LIN {X 0,Y 79.214,Z 378.176,A -85,B 0,C 180,E1 -30939.921,E2 -30939.921} C_VEL
LIN {X 0,Y 81.535,Z 365.2,A -85,B 0,C 180,E1 -30940.229,E2 -30940.229} C_VEL
LIN {X 0,Y 82.563,Z 356.649,A -85,B 0,C 180,E1 -30940.524,E2 -30940.524} C_VEL
LIN {X 0,Y 82.095,Z 354.312,A -85,B 0,C 180,E1 -30944.218,E2 -30944.218} C_VEL
LIN {X 0,Y 81.886,Z 351.905,A -85,B 0,C 180,E1 -30950.139,E2 -30950.139} C_VEL
LIN {X 0,Y 81.95,Z 352.015,A -85,B 0,C 180,E1 -30953.705,E2 -30953.705} C_VEL
LIN {X 0,Y 82.216,Z 354.524,A -85,B 0,C 180,E1 -30958.491,E2 -30958.491} C_VEL
LIN {X 0,Y 82.607,Z 356.769,A -85,B 0,C 180,E1 -30961.538,E2 -30961.538} C_VEL
LIN {X 0,Y 80.054,Z 374.634,A -85,B 0,C 180,E1 -30961.987,E2 -30961.987} C_VEL
LIN {X 0,Y 76.93,Z 387.122,A -85,B 0,C 180,E1 -30962.346,E2 -30962.346} C_VEL
LIN {X 0,Y 72.584,Z 399.313,A -85,B 0,C 180,E1 -30963.156,E2 -30963.156} C_VEL
LIN {X 0,Y 66.925,Z 411.041,A -85,B 0,C 180,E1 -30963.978,E2 -30963.978} C_VEL
LIN {X 0,Y 62.589,Z 418.476,A -85,B 0,C 180,E1 -30964.782,E2 -30964.782} C_VEL
LIN {X 0,Y 55.7,Z 428.368,A -85,B 0,C 180,E1 -30966.498,E2 -30966.498} C_VEL
LIN {X 0,Y 49.71,Z 435.606,A -85,B 0,C 180,E1 -30968.267,E2 -30968.267} C_VEL
LIN {X 0,Y 41.286,Z 444.313,A -85,B 0,C 180,E1 -30971.836,E2 -30971.836} C_VEL
LIN {X 0,Y 31.466,Z 452.724,A -85,B 0,C 180,E1 -30978.346,E2 -30978.346} C_VEL
LIN {X 0,Y 22.335,Z 459.473,A -85,B 0,C 180,E1 -30990.091,E2 -30990.091} C_VEL
LIN {X 0,Y 14.338,Z 465.618,A -85,B 0,C 180,E1 -31020.66,E2 -31020.66} C_VEL
LIN {X 0,Y 12.95,Z 468.35,A -85,B 0,C 180,E1 -31050.01,E2 -31050.01} C_VEL
LIN {X 0,Y 14.464,Z 470.587,A -85,B 0,C 180,E1 -31079.082,E2 -31079.082} C_VEL
LIN {X 0,Y 18.52,Z 472.391,A -85,B 0,C 180,E1 -31099.384,E2 -31099.384} C_VEL
LIN {X 0,Y 30.065,Z 474.714,A -85,B 0,C 180,E1 -31119.245,E2 -31119.245} C_VEL
LIN {X 0,Y 43.205,Z 475.536,A -85,B 0,C 180,E1 -31127.436,E2 -31127.436} C_VEL
LIN {X 0,Y 49.975,Z 475.374,A -85,B 0,C 180,E1 -31129.886,E2 -31129.886} C_VEL
LIN {X 0,Y 52.842,Z 475.146,A -85,B 0,C 180,E1 -31132.323,E2 -31132.323} C_VEL
LIN {X 0,Y 42.273,Z 475.423,A -85,B 0,C 180,E1 -31136.005,E2 -31136.005} C_VEL
LIN {X 0,Y 34.947,Z 475.052,A -85,B 0,C 180,E1 -31139.948,E2 -31139.948} C_VEL
LIN {X 0,Y 28.242,Z 474.29,A -85,B 0,C 180,E1 -31145.454,E2 -31145.454} C_VEL
LIN {X 0,Y 18.34,Z 472.097,A -85,B 0,C 180,E1 -31162.424,E2 -31162.424} C_VEL
LIN {X 0,Y 12.711,Z 469.162,A -85,B 0,C 180,E1 -31196.422,E2 -31196.422} C_VEL
LIN {X 0,Y 14.539,Z 464.821,A -85,B 0,C 180,E1 -31245.295,E2 -31245.295} C_VEL
LIN {X 0,Y 21.792,Z 459.578,A -85,B 0,C 180,E1 -31270.158,E2 -31270.158} C_VEL
LIN {X 0,Y 24.176,Z 457.887,A -85,B 0,C 180,E1 -31274.413,E2 -31274.413} C_VEL
LIN {X 0,Y 28.142,Z 454.814,A -85,B 0,C 180,E1 -31281.291,E2 -31281.291} C_VEL
LIN {X 0,Y 34.16,Z 449.309,A -85,B 0,C 180,E1 -31291.795,E2 -31291.795} C_VEL
LIN {X 0,Y 40.474,Z 443.166,A -85,B 0,C 180,E1 -31298.966,E2 -31298.966} C_VEL
LIN {X 0,Y 44.545,Z 439.087,A -85,B 0,C 180,E1 -31300.86,E2 -31300.86} C_VEL
LIN {X 0,Y 53.478,Z 429.1,A -85,B 0,C 180,E1 -31302.312,E2 -31302.312} C_VEL
LIN {X 0,Y 61.443,Z 418.069,A -85,B 0,C 180,E1 -31303.319,E2 -31303.319} C_VEL
LIN {X 0,Y 67.627,Z 407.259,A -85,B 0,C 180,E1 -31303.998,E2 -31303.998} C_VEL
LIN {X 0,Y 72.904,Z 395.421,A -85,B 0,C 180,E1 -31304.574,E2 -31304.574} C_VEL
LIN {X 0,Y 77.246,Z 382.161,A -85,B 0,C 180,E1 -31304.973,E2 -31304.973} C_VEL
LIN {X 0,Y 79.976,Z 369.173,A -85,B 0,C 180,E1 -31305.151,E2 -31305.151} C_VEL
LIN {X 0,Y 81.055,Z 361.14,A -85,B 0,C 180,E1 -31305.371,E2 -31305.371} C_VEL
LIN {X 0,Y 80.991,Z 358.94,A -85,B 0,C 180,E1 -31310.659,E2 -31310.659} C_VEL
LIN {X 0,Y 81.008,Z 359.111,A -85,B 0,C 180,E1 -31312.98,E2 -31312.98} C_VEL
LIN {X 0,Y 81.091,Z 361.038,A -85,B 0,C 180,E1 -31316.663,E2 -31316.663} C_VEL
LIN {X 0,Y 78.773,Z 375.942,A -85,B 0,C 180,E1 -31316.949,E2 -31316.949} C_VEL
LIN {X 0,Y 75.741,Z 387.538,A -85,B 0,C 180,E1 -31317.105,E2 -31317.105} C_VEL
LIN {X 0,Y 71.058,Z 400.138,A -85,B 0,C 180,E1 -31317.612,E2 -31317.612} C_VEL
LIN {X 0,Y 65.05,Z 412.155,A -85,B 0,C 180,E1 -31317.891,E2 -31317.891} C_VEL
LIN {X 0,Y 57.993,Z 423.301,A -85,B 0,C 180,E1 -31318.699,E2 -31318.699} C_VEL
LIN {X 0,Y 50.951,Z 432.35,A -85,B 0,C 180,E1 -31319.863,E2 -31319.863} C_VEL
LIN {X 0,Y 43.541,Z 440.271,A -85,B 0,C 180,E1 -31321.038,E2 -31321.038} C_VEL
LIN {X 0,Y 33.461,Z 449.191,A -85,B 0,C 180,E1 -31323.983,E2 -31323.983} C_VEL
LIN {X 0,Y 23.116,Z 456.621,A -85,B 0,C 180,E1 -31328.892,E2 -31328.892} C_VEL
LIN {X 0,Y 14.813,Z 461.66,A -85,B 0,C 180,E1 -31338.424,E2 -31338.424} C_VEL
LIN {X 0,Y 6.659,Z 466.511,A -85,B 0,C 180,E1 -31378.171,E2 -31378.171} C_VEL
LIN {X 0,Y 6.772,Z 469.093,A -85,B 0,C 180,E1 -31441.281,E2 -31441.281} C_VEL
LIN {X 0,Y 14.906,Z 472.022,A -85,B 0,C 180,E1 -31480.58,E2 -31480.58} C_VEL
LIN {X 0,Y 21.514,Z 473.472,A -85,B 0,C 180,E1 -31488.55,E2 -31488.55} C_VEL
LIN {X 0,Y 23.942,Z 473.852,A -85,B 0,C 180,E1 -31492.249,E2 -31492.249} C_VEL
LIN {X 0,Y 14.068,Z 471.73,A -85,B 0,C 180,E1 -31502.166,E2 -31502.166} C_VEL
LIN {X 0,Y 5.569,Z 468.397,A -85,B 0,C 180,E1 -31550.848,E2 -31550.848} C_VEL
LIN {X 0,Y 10.326,Z 463.944,A -85,B 0,C 180,E1 -31632.875,E2 -31632.875} C_VEL
LIN {X 0,Y 20.972,Z 457.864,A -85,B 0,C 180,E1 -31650.55,E2 -31650.55} C_VEL
LIN {X 0,Y 30.66,Z 451.233,A -85,B 0,C 180,E1 -31656.465,E2 -31656.465} C_VEL
LIN {X 0,Y 40.702,Z 442.81,A -85,B 0,C 180,E1 -31659.846,E2 -31659.846} C_VEL
LIN {X 0,Y 44.545,Z 439.087,A -85,B 0,C 180,E1 -31660.86,E2 -31660.86} C_VEL
LIN {X 0,Y 48.458,Z 434.878,A -85,B 0,C 180,E1 -31662.371,E2 -31662.371} C_VEL
LIN {X 0,Y 54.291,Z 427.659,A -85,B 0,C 180,E1 -31666.195,E2 -31666.195} C_VEL
LIN {X 0,Y 59.756,Z 419.952,A -85,B 0,C 180,E1 -31669.291,E2 -31669.291} C_VEL
LIN {X 0,Y 62.931,Z 414.933,A -85,B 0,C 180,E1 -31669.948,E2 -31669.948} C_VEL
LIN {X 0,Y 68.666,Z 404.345,A -85,B 0,C 180,E1 -31670.091,E2 -31670.091} C_VEL
LIN {X 0,Y 73.843,Z 391.921,A -85,B 0,C 180,E1 -31670.162,E2 -31670.162} C_VEL
LIN {X 0,Y 77.709,Z 378.813,A -85,B 0,C 180,E1 -31670.218,E2 -31670.218} C_VEL
LIN {X 0,Y 79.946,Z 366.975,A -85,B 0,C 180,E1 -31670.23,E2 -31670.23} C_VEL
LIN {X 0,Y 80.038,Z 366.349,A -85,B 0,C 180,E1 -31670.553,E2 -31670.553} C_VEL
LIN {X 0,Y 80.094,Z 365.965,A -85,B 0,C 180,E1 -31671.678,E2 -31671.678} C_VEL
LIN {X 0,Y 77.931,Z 377.897,A -85,B 0,C 180,E1 -31671.747,E2 -31671.747} C_VEL
LIN {X 0,Y 74.454,Z 390.128,A -85,B 0,C 180,E1 -31671.777,E2 -31671.777} C_VEL
LIN {X 0,Y 70.105,Z 401.23,A -85,B 0,C 180,E1 -31671.861,E2 -31671.861} C_VEL
LIN {X 0,Y 64.817,Z 411.708,A -85,B 0,C 180,E1 -31671.64,E2 -31671.64} C_VEL
LIN {X 0,Y 57.707,Z 422.936,A -85,B 0,C 180,E1 -31671.683,E2 -31671.683} C_VEL
LIN {X 0,Y 49.7,Z 433.016,A -85,B 0,C 180,E1 -31671.813,E2 -31671.813} C_VEL
LIN {X 0,Y 42.614,Z 440.46,A -85,B 0,C 180,E1 -31671.677,E2 -31671.677} C_VEL
LIN {X 0,Y 31.956,Z 449.628,A -85,B 0,C 180,E1 -31671.724,E2 -31671.724} C_VEL
LIN {X 0,Y 21.347,Z 456.964,A -85,B 0,C 180,E1 -31670.958,E2 -31670.958} C_VEL
LIN {X 0,Y 21.392,Z 456.933,A -85,B 0,C 180,E1 -31670.232,E2 -31670.232} C_VEL
LIN {X 0,Y 32.126,Z 449.489,A -85,B 0,C 180,E1 -31669.85,E2 -31669.85} C_VEL
LIN {X 0,Y 41.569,Z 441.425,A -85,B 0,C 180,E1 -31669.987,E2 -31669.987} C_VEL
LIN {X 0,Y 50.845,Z 431.714,A -85,B 0,C 180,E1 -31669.998,E2 -31669.998} C_VEL
LIN {X 0,Y 58.884,Z 421.206,A -85,B 0,C 180,E1 -31669.94,E2 -31669.94} C_VEL
LIN {X 0,Y 62.931,Z 414.933,A -85,B 0,C 180,E1 -31669.948,E2 -31669.948} C_VEL
LIN {X 0,Y 66.635,Z 415.981,A -85,B 0,C 180,E1 -31669.987,E2 -31669.987} C_VEL
LIN {X 0,Y 66.635,Z 600,A -85,B 0,C 180,E1 -31669.987,E2 -31669.987} C_VEL
LIN {X 0,Y 66.635,Z 600,A -85,B 0,C 180,E1 -31669.987,E2 -31669.987}

QRS_NEXT_CUT()

QRS_NEXT()
QRS_HOME()

END
